// TIA Portal project "sayici_ile_motor_çalistirma" (V18)

(* hardware
DEVICE "S7-1200 station_1"  S7-1200 Station
   slot 0: "Rack_0"  S7-1200 Rack  Rack  V1.0
   slot 1: "PLC_1"  CPU 1214C AC/DC/Rly  6ES7 214-1BG40-0XB0  V4.6
*)

// ===== PLC "PLC_1"  CPU 1214C AC/DC/Rly =====

VAR_GLOBAL   // PLC tag table "Default tag table"
   "START" AT %I0.0 : Bool;
   "STOP" AT %I0.1 : Bool;
   "MOTOR" AT %Q0.0 : Bool;
   "Tag_1" AT %M100.0 : Bool;
   "Tag_2" AT %MW0 : Int;
   "Tag_3" AT %M100.1 : Bool;
END_VAR

// folder: System blocks/Program resources

DATA_BLOCK "C1"   // DB1
{ S7_Optimized_Access := 'TRUE' }
AUTHOR : Simatic
FAMILY : IEC
NAME : CNTR
VERSION : 1.0
// stored: InstanceOfName IEC_COUNTER
"IEC_COUNTER"
BEGIN
END_DATA_BLOCK

DATA_BLOCK "C2"   // DB2
{ S7_Optimized_Access := 'TRUE' }
AUTHOR : Simatic
FAMILY : IEC
NAME : CNTR
VERSION : 1.0
// stored: InstanceOfName IEC_COUNTER
"IEC_COUNTER"
BEGIN
END_DATA_BLOCK

// folder: (top level)

ORGANIZATION_BLOCK "Main"   // OB1, LAD, ProgramCycle
TITLE = "Main Program Sweep (Cycle)"
{ S7_Optimized_Access := 'TRUE' }
VERSION : 0.1
   VAR_INPUT
      Initial_Call : Bool;   // Initial call of this OB
      Remanence : Bool;   // =True, if remanent data are available
   END_VAR
   VAR_TEMP   // added for the SCL form of the ladder/FBD networks
      _w1 : Bool;
   END_VAR
BEGIN

REGION Network 1
   // ilk iki network, start ve stop butonları ile motor çalıştırmadır.
   // Sonrakiler ise kesikli ve sürekli çalıştırma örnekleri
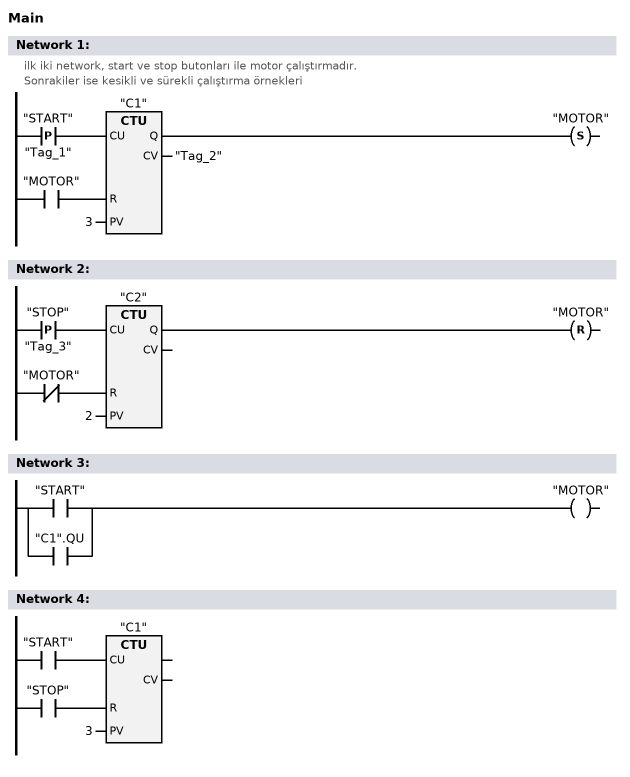
   #_w1 := "START" AND NOT "Tag_1";   // rising edge of "START"
   "Tag_1" := "START";
   "C1".CTU(CU := #_w1, R := "MOTOR", PV := 3, CV => "Tag_2");
   IF "C1".Q THEN "MOTOR" := TRUE; END_IF;
END_REGION

REGION Network 2
   #_w1 := "STOP" AND NOT "Tag_3";   // rising edge of "STOP"
   "Tag_3" := "STOP";
   "C2".CTU(CU := #_w1, R := NOT "MOTOR", PV := 2);
   IF "C2".Q THEN "MOTOR" := FALSE; END_IF;
END_REGION

REGION Network 3
   RUNG wire#powerrail
      Contact( "START" )
      wire#w1
      Coil( "MOTOR" )
   END_RUNG
   RUNG wire#powerrail
      Contact( "C1".QU )
   END_RUNG wire#w1
   // the same network as SCL:
   "MOTOR" := "START" OR "C1".QU;
END_REGION

REGION Network 4
   "C1".CTU(CU := "START", R := "STOP", PV := 3);
END_REGION
END_ORGANIZATION_BLOCK